FUNCTION_BLOCK Station IMPLEMENTS IStation
VAR_INPUT
END_VAR
VAR_OUTPUT
END_VAR
VAR
	_Clear : BOOL;
	_Complete : BOOL;
	_Operating : BOOL;
	_Ready : BOOL;
	_Positions : ARRAY[1..4] OF MC_LREAL;
	NumberOfPositions : INT;
	AssignedPositions : INT := 1;
	StationMovers : INT;
	_OperationTime : TIME := T#1S;
	Operation : ton;
	_HasMover : BOOL;
END_VAR

IF _HasMover THEN
	_Operating := TRUE;
	_Clear := FALSE;
	_Ready := FALSE;
	Operation.IN := TRUE;
	IF Operation.Q THEN
		_Complete := TRUE;
		IF StationMovers = 0 THEN
			_HasMover := FALSE;
			Operation.IN := FALSE;
		END_IF
	END_IF
ELSE
	_Complete := FALSE;
	_Clear := TRUE;
	_Operating := FALSE;
	_Ready := TRUE;
END_IF

Operation(PT := _OperationTime);

{warning 'add method implementation '}
METHOD HasMover : BOOL
StationMovers := StationMovers + 1;
IF StationMovers = NumberOfPositions THEN
	_HasMover := TRUE;
END_IF
END_METHOD

{warning 'add method implementation '}
METHOD IsClear : BOOL
IsClear := _Clear;
END_METHOD

{warning 'add method implementation '}
METHOD isComplete : BOOL
isComplete := _Complete;
END_METHOD

{warning 'add method implementation '}
METHOD IsOperating : BOOL
IsOperating := _Operating;
END_METHOD

{warning 'add method implementation '}
METHOD IsReady : BOOL
IsReady := _Ready;
END_METHOD

METHOD MoverAway : BOOL
VAR_INPUT
END_VAR
StationMovers := StationMovers - 1;
END_METHOD

{warning 'add property implementation'}
PROPERTY Position : MC_LREAL
GET
Position := _Positions[AssignedPositions];
AssignedPositions := AssignedPositions + 1;
IF AssignedPositions > NumberOfPositions THEN
	AssignedPositions := 1;
END_IF
END_GET
SET
IF NumberOfPositions < 5 THEN
	NumberOfPositions := NumberOfPositions + 1;
	_Positions[NumberOfPositions] := Position;
END_IF
END_SET
END_PROPERTY

PROPERTY TempPropTime : time
GET
TempPropTime := _OperationTime;
END_GET
SET
_OperationTime := TempPropTime;
END_SET
END_PROPERTY

END_FUNCTION_BLOCK

(* stored: Version 1.1.0.1, ProductVersion 3.1.4024.11
   POU Station: Id {15da8106-0d22-4ca5-af9c-31c3d97b8668}, SpecialFunc None
   Method HasMover: Id {1cb719ab-8b5a-456f-a91b-48331f9d0dc2}
   Method IsClear: Id {76a4496f-67c0-45fc-9e15-a528954fd797}
   Method isComplete: Id {e952f541-8c98-4290-8bef-72b636ded12c}
   Method IsOperating: Id {46f6a6eb-2d48-45d2-a61c-982a5af29ec7}
   Method IsReady: Id {72424547-540c-4f0b-8c61-f3533ca0048c}
   Method MoverAway: Id {5bac361c-272f-42b5-96ba-9a558f55b3c0}
   Property Position: Id {4a10e32c-305e-441b-9332-8642baafa7cc}
   Get Get: Id {6760ec00-0cdd-4667-9f90-fd015738ea5e}
   Set Set: Id {825e159a-d125-4194-a2b1-af8249a79ce1}
   Property TempPropTime: Id {e0ccb7b2-ab4d-4401-a6ea-ec63ab2ed8d6}
   Get Get: Id {d09bc174-9f05-4e5a-bc80-e72251b6839f}
   Set Set: Id {cefc9927-2f03-41f9-b855-e64e1bbf9aa6} *)
